RoboDK station: practica1DosCubos.rdk

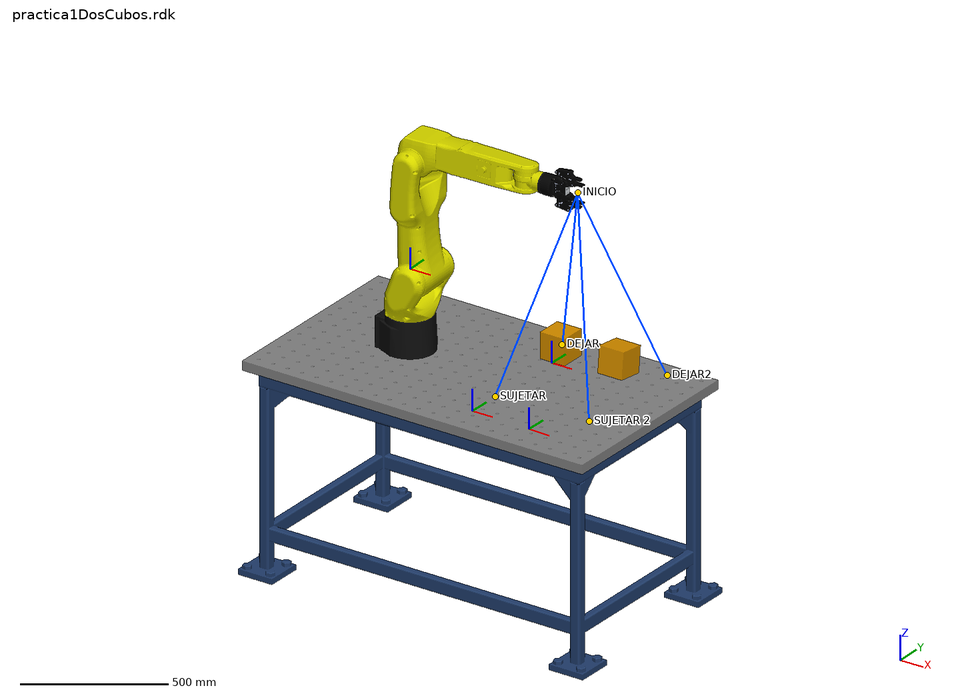
[picture v0: the station drawn from its stored meshes, robots at their saved joint values, targets as dots, program paths as lines]
Station practica1DosCubos (saved by RoboDK 6.0.0). Poses are relative to the parent item; angles as X-Y-Z fixed-axis rotations.
  - object Table 1400x800x800mm at (0, 0, 0) mm, size 1420 x 820 x 800 mm, geometry from Table-1400x800x800mm.sld
  - frame Fanuc LR Mate 200iD/7L Base at (70.2, 3.67, 297.49) mm, rotated rx 0.7 ry 0.59 rz 1.98 deg
    - robot Fanuc LR Mate 200iD/7L: 6 axes, payload 7 kg, reach 911 mm, repeatability 0.01 mm, weight 27 kg
        modified DH rows (alpha deg, a mm, theta deg, d mm): 0, 0, 0, 330; -90, 50, -90, 0; 0, 440, 0, 0; -90, 35, 0, 420; 90, 0, 0, 0; -90, 0, 0, 80
        base shift (0, 0, -330) mm
        joint limits [-180, -100, -150, -190, -125, -360] to [180, 145, 280, 190, 125, 360]; home [0, 0, 0, 0, 0, 0]; saved at [0.03, -0.915, -0.003, -85.15, 0.023, 85.15]
      - tool RobotiQ 2F-85 Gripper (Open), TCP at (0, 0, 130) mm, size 147.4 x 75 x 146.8 mm
      - tool RobotiQ 2F-85 Gripper (Closed), TCP at (0, 0, 130) mm, size 134.4 x 75 x 157.6 mm
  - frame PICK at (538.36, -298.62, 16) mm
    - target INICIO (Cartesian target) at (209.42, 320.17, 749.47) mm, rotated rx -129.84 ry -89.09 rz -48.18 deg; joints [0, 0, 0, 0, 0, 0] of Fanuc LR Mate 200iD/7L
    - target SUJETAR (Cartesian target) at (56.61, 52.29, 49.23) mm, rotated rx -131.44 ry -89.06 rz -46.58 deg; joints [-41.305, 63.462, -99.313, 41.679, 96.948, 6.177] of Fanuc LR Mate 200iD/7L
    - target DEJAR (Cartesian target) at (21.12, 496.71, 56.53) mm, rotated rx -129.83 ry -89.09 rz -48.19 deg; joints [31.235, 65.277, -110.295, -32.887, 107.252, -10.856] of Fanuc LR Mate 200iD/7L
  - frame PLACE at (547.88, 151.77, 19.41) mm
  - frame PICK2 at (767.97, -293.83, 10.18) mm
    - target SUJETAR 2 (Cartesian target) at (194.84, 74.23, 55.52) mm, rotated rx -124.22 ry -89.08 rz -48.14 deg; joints [-31.472, 63.365, -83.548, -142.696, -84.857, 176.092] of Fanuc LR Mate 200iD/7L
    - target DEJAR2 (Cartesian target) at (202.5, 523.31, 48.82) mm, rotated rx 103.93 ry -84.17 rz 83.57 deg; joints [20.376, 64.03, -86.977, -14.975, 86.195, 7.195] of Fanuc LR Mate 200iD/7L
  - program Prog1 (15 instructions, listed below)
  - object Cube 100mm at (499.93, 153.08, 22.32) mm, rotated rx 0 ry -0.03 rz 0 deg, size 100 x 100 x 100 mm, geometry from Cube-100mm.sld
  - object Cube 100mm at (734.78, 154.79, 33.63) mm, rotated rx -6.48 ry -0.01 rz -0.1 deg, size 100 x 100 x 100 mm, geometry from Cube-100mm.sld
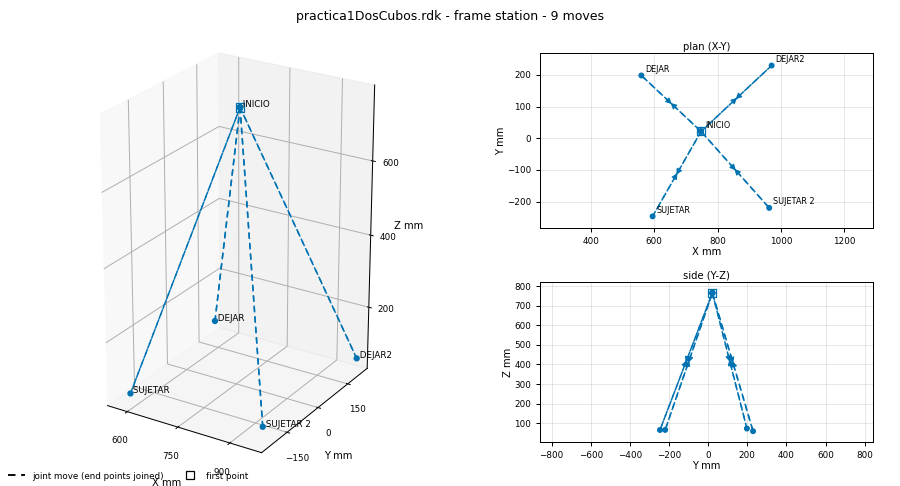
[picture p0: tool path of practica1DosCubos.rdk in frame station, 9 of 9 moves have a stored position in this frame; points joined in program order, loops and branches not executed]

--- program Prog1 (robot Fanuc LR Mate 200iD/7L) ---
  Est. Ref.: PICK
  Est. herr: RobotiQ 2F-85 Gripper (Open)
  MoveJ (INICIO)
  MoveJ (SUJETAR)
  Adjuntar a RobotiQ 2F-85 Gripper (Open)
  MoveJ (INICIO)
  MoveJ (DEJAR)
  Separar de RobotiQ 2F-85 Gripper (Open)
  MoveJ (INICIO)
  MoveJ (SUJETAR 2)
  Adjuntar a RobotiQ 2F-85 Gripper (Open)
  MoveJ (INICIO)
  MoveJ (DEJAR2)
  Separar de RobotiQ 2F-85 Gripper (Open)
  MoveJ (INICIO)
